// TIA Portal V17 export
// export: Created 2023-12-22T15:05:31.7217918Z, ExportSetting WithDefaults, DisplayName Totally Integrated Automation Portal, DisplayVersion V17, DisplayName TIA Portal Openness, DisplayVersion V17, DisplayName TIA Portal Version Control Interface, DisplayVersion V17, DisplayName STEP 7 Professional, DisplayVersion V17, DisplayName STEP 7 Safety, DisplayVersion V17, DisplayName WinCC Advanced, DisplayVersion V17
FUNCTION_BLOCK "FB_DRV_Start"   // FB100, LAD
{ S7_Optimized_Access := 'TRUE' }
VERSION : 0.1
// stored: AutoNumber false, IsIECCheckEnabled false, IsRetainMemResEnabled false, MemoryReserve 100, SetENOAutomatically false, UDAEnableTagReadback false
   VAR
      last_01s : Int;
      last_05s : Int;
      last_1s : Int;
      last_5s : Int;
      last_10s : Int;
      last_30s : Int;
      last_1m : Int;
      last_5m : Int;
      last_10m : Int;
      last_30m : Int;
      last_1h : Int;
      last_1_day : Int;
      last_1_week : Int;
      last_1_month : Int;
      last_s1 : Int;
      last_s2 : Int;
      "1h_minutes" { S7_SetPoint := 'True'} : Int;
      "1_day_hour" { S7_SetPoint := 'True'} : Int;
      "1_day_minutes" { S7_SetPoint := 'True'} : Int;
      "1_week_weekday" { S7_SetPoint := 'True'} : Int := 1;
      "1_week_hour" { S7_SetPoint := 'True'} : Int;
      "1_week_minutes" { S7_SetPoint := 'True'} : Int;
      "1_month_date" { S7_SetPoint := 'True'} : Int := 1;
      "1_month_hour" { S7_SetPoint := 'True'} : Int;
      "1_month_minutes" { S7_SetPoint := 'True'} : Int;
      s1_hour : Int := 8;
      s1_minutes : Int;
      s2_hour : Int := 20;
      s2_minutes : Int;
      pos : Array[0..15] of Bool;
      Error : Word;
      x { S7_SetPoint := 'True'} : "Protection";
   END_VAR
   VAR_TEMP
      cnt_01s : Int;
      cnt_5s : Int;
      cnt_10s : Int;
      cnt_30s : Int;
      cnt_5m : Int;
      cnt_10m : Int;
      cnt_30m : Int;
   END_VAR
   VAR_TEMP   // added for the SCL form of the ladder/FBD networks
      _w1 : Bool;
      _w2 : Bool;
   END_VAR
BEGIN

REGION Network 1: Обработчик системного времени
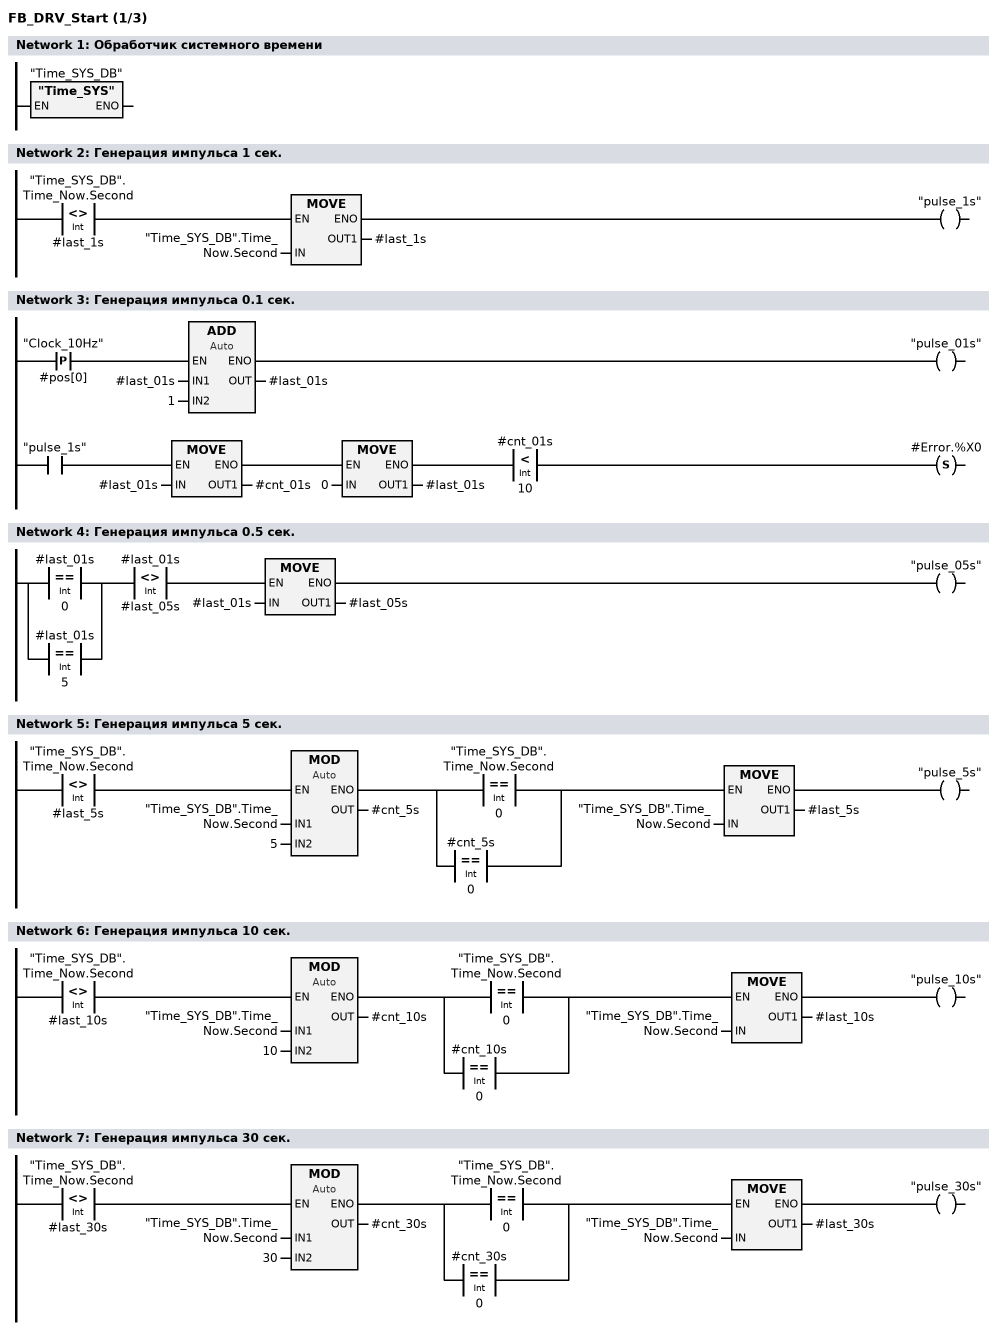
   RUNG wire#powerrail
      "Time_SYS_DB"()
   END_RUNG
   // the same network as SCL:
   "Time_SYS_DB"();   // "Time_SYS"
END_REGION

REGION Network 2: Генерация импульса 1 сек.
   RUNG wire#powerrail
      { S7_Templates := "SrcType := Int" } NE_Contact(in1 := "Time_SYS_DB".Time_Now.Second, in2 := #last_1s)
      Move(in := "Time_SYS_DB".Time_Now.Second, out1 => #last_1s)
      Coil( "pulse_1s" )
   END_RUNG
   // the same network as SCL:
   #_w1 := "Time_SYS_DB".Time_Now.Second <> #last_1s;
   IF #_w1 THEN #last_1s := "Time_SYS_DB".Time_Now.Second; END_IF;
   "pulse_1s" := #_w1;
END_REGION

REGION Network 3: Генерация импульса 0.1 сек.
   RUNG wire#powerrail
      P_Contact(operand := "Clock_10Hz", bit := #pos[0])
      Add(in1 := #last_01s, in2 := 1, out => #last_01s)
      Coil( "pulse_01s" )
   END_RUNG
   RUNG wire#powerrail
      Contact( "pulse_1s" )
      Move(in := #last_01s, out1 => #cnt_01s)
      Move(in := 0, out1 => #last_01s)
      { S7_Templates := "SrcType := Int" } LT_Contact(in1 := #cnt_01s, in2 := 10)
      S_Coil( #Error.%X0 )
   END_RUNG
   // the same network as SCL:
   #_w1 := "Clock_10Hz" AND NOT #pos[0];   // rising edge of "Clock_10Hz"
   #pos[0] := "Clock_10Hz";
   IF #_w1 THEN #last_01s := #last_01s + 1; END_IF;
   "pulse_01s" := #_w1;
   IF "pulse_1s" THEN
       #cnt_01s := #last_01s;
       #last_01s := 0;
   END_IF;
   IF "pulse_1s" AND (#cnt_01s < 10) THEN #Error.%X0 := TRUE; END_IF;
END_REGION

REGION Network 4: Генерация импульса 0.5 сек.
   RUNG wire#powerrail
      { S7_Templates := "SrcType := Int" } EQ_Contact(in1 := #last_01s, in2 := 0)
      wire#w1
      { S7_Templates := "SrcType := Int" } NE_Contact(in1 := #last_01s, in2 := #last_05s)
      Move(in := #last_01s, out1 => #last_05s)
      Coil( "pulse_05s" )
   END_RUNG
   RUNG wire#powerrail
      { S7_Templates := "SrcType := Int" } EQ_Contact(in1 := #last_01s, in2 := 5)
   END_RUNG wire#w1
   // the same network as SCL:
   #_w1 := ((#last_01s = 0) OR (#last_01s = 5)) AND (#last_01s <> #last_05s);
   IF #_w1 THEN #last_05s := #last_01s; END_IF;
   "pulse_05s" := #_w1;
END_REGION

REGION Network 5: Генерация импульса 5 сек.
   RUNG wire#powerrail
      { S7_Templates := "SrcType := Int" } NE_Contact(in1 := "Time_SYS_DB".Time_Now.Second, in2 := #last_5s)
      Mod(in1 := "Time_SYS_DB".Time_Now.Second, in2 := 5, out => #cnt_5s)
      wire#w1
      { S7_Templates := "SrcType := Int" } EQ_Contact(in1 := "Time_SYS_DB".Time_Now.Second, in2 := 0)
      wire#w2
      Move(in := "Time_SYS_DB".Time_Now.Second, out1 => #last_5s)
      Coil( "pulse_5s" )
   END_RUNG
   RUNG wire#w1
      { S7_Templates := "SrcType := Int" } EQ_Contact(in1 := #cnt_5s, in2 := 0)
   END_RUNG wire#w2
   // the same network as SCL:
   #_w1 := "Time_SYS_DB".Time_Now.Second <> #last_5s;
   IF #_w1 THEN #cnt_5s := "Time_SYS_DB".Time_Now.Second MOD 5; END_IF;
   #_w2 := #_w1 AND (("Time_SYS_DB".Time_Now.Second = 0) OR (#cnt_5s = 0));
   IF #_w2 THEN #last_5s := "Time_SYS_DB".Time_Now.Second; END_IF;
   "pulse_5s" := #_w2;
END_REGION

REGION Network 6: Генерация импульса 10 сек.
   RUNG wire#powerrail
      { S7_Templates := "SrcType := Int" } NE_Contact(in1 := "Time_SYS_DB".Time_Now.Second, in2 := #last_10s)
      Mod(in1 := "Time_SYS_DB".Time_Now.Second, in2 := 10, out => #cnt_10s)
      wire#w1
      { S7_Templates := "SrcType := Int" } EQ_Contact(in1 := "Time_SYS_DB".Time_Now.Second, in2 := 0)
      wire#w2
      Move(in := "Time_SYS_DB".Time_Now.Second, out1 => #last_10s)
      Coil( "pulse_10s" )
   END_RUNG
   RUNG wire#w1
      { S7_Templates := "SrcType := Int" } EQ_Contact(in1 := #cnt_10s, in2 := 0)
   END_RUNG wire#w2
   // the same network as SCL:
   #_w1 := "Time_SYS_DB".Time_Now.Second <> #last_10s;
   IF #_w1 THEN #cnt_10s := "Time_SYS_DB".Time_Now.Second MOD 10; END_IF;
   #_w2 := #_w1 AND (("Time_SYS_DB".Time_Now.Second = 0) OR (#cnt_10s = 0));
   IF #_w2 THEN #last_10s := "Time_SYS_DB".Time_Now.Second; END_IF;
   "pulse_10s" := #_w2;
END_REGION

REGION Network 7: Генерация импульса 30 сек.
   RUNG wire#powerrail
      { S7_Templates := "SrcType := Int" } NE_Contact(in1 := "Time_SYS_DB".Time_Now.Second, in2 := #last_30s)
      Mod(in1 := "Time_SYS_DB".Time_Now.Second, in2 := 30, out => #cnt_30s)
      wire#w1
      { S7_Templates := "SrcType := Int" } EQ_Contact(in1 := "Time_SYS_DB".Time_Now.Second, in2 := 0)
      wire#w2
      Move(in := "Time_SYS_DB".Time_Now.Second, out1 => #last_30s)
      Coil( "pulse_30s" )
   END_RUNG
   RUNG wire#w1
      { S7_Templates := "SrcType := Int" } EQ_Contact(in1 := #cnt_30s, in2 := 0)
   END_RUNG wire#w2
   // the same network as SCL:
   #_w1 := "Time_SYS_DB".Time_Now.Second <> #last_30s;
   IF #_w1 THEN #cnt_30s := "Time_SYS_DB".Time_Now.Second MOD 30; END_IF;
   #_w2 := #_w1 AND (("Time_SYS_DB".Time_Now.Second = 0) OR (#cnt_30s = 0));
   IF #_w2 THEN #last_30s := "Time_SYS_DB".Time_Now.Second; END_IF;
   "pulse_30s" := #_w2;
END_REGION

REGION Network 8: Генерация импульса 1 мин.
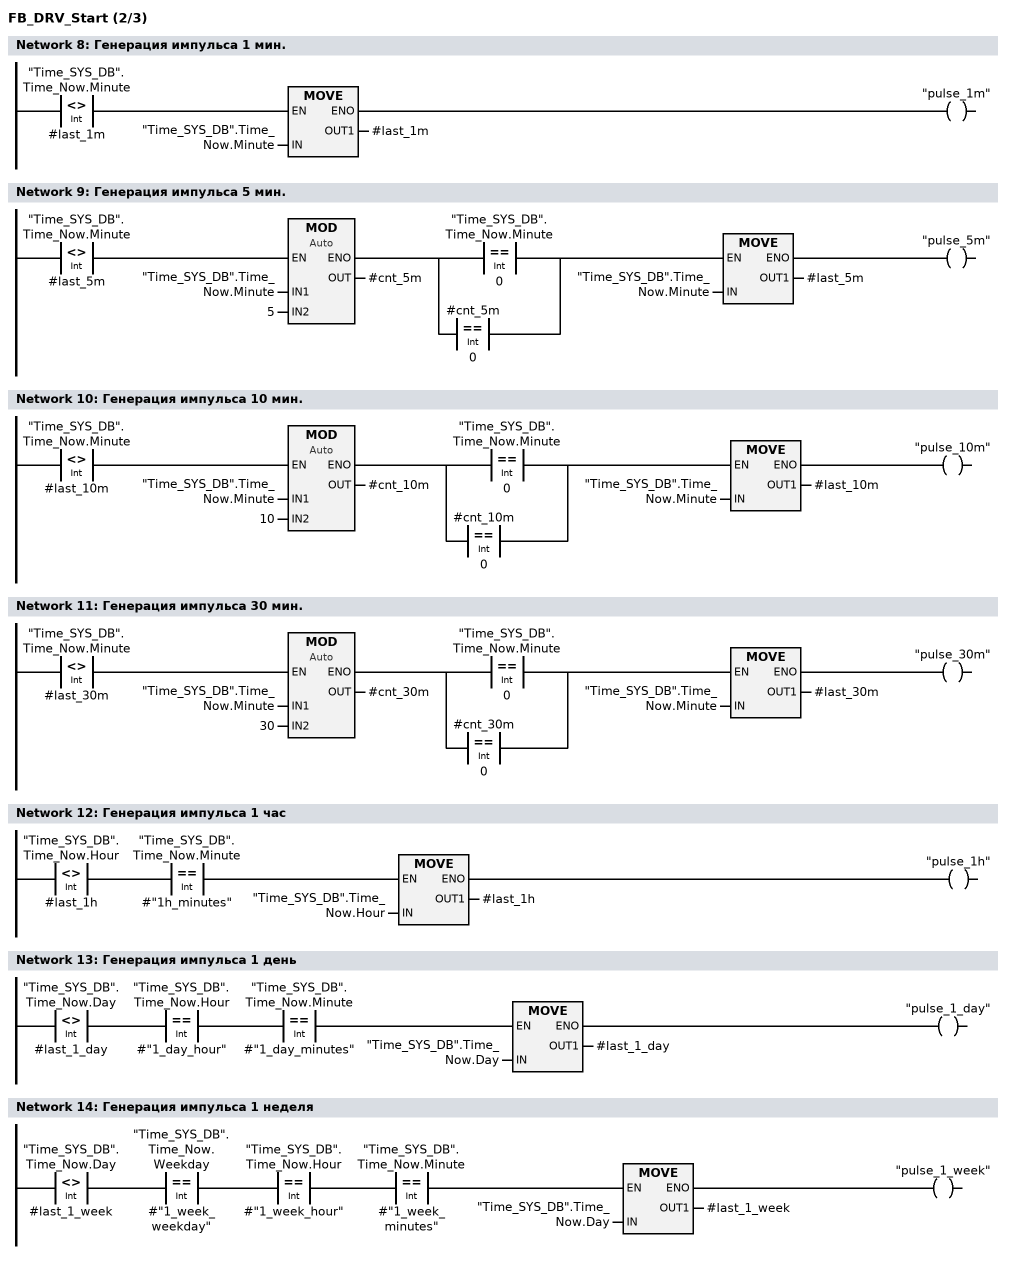
   RUNG wire#powerrail
      { S7_Templates := "SrcType := Int" } NE_Contact(in1 := "Time_SYS_DB".Time_Now.Minute, in2 := #last_1m)
      Move(in := "Time_SYS_DB".Time_Now.Minute, out1 => #last_1m)
      Coil( "pulse_1m" )
   END_RUNG
   // the same network as SCL:
   #_w1 := "Time_SYS_DB".Time_Now.Minute <> #last_1m;
   IF #_w1 THEN #last_1m := "Time_SYS_DB".Time_Now.Minute; END_IF;
   "pulse_1m" := #_w1;
END_REGION

REGION Network 9: Генерация импульса 5 мин.
   RUNG wire#powerrail
      { S7_Templates := "SrcType := Int" } NE_Contact(in1 := "Time_SYS_DB".Time_Now.Minute, in2 := #last_5m)
      Mod(in1 := "Time_SYS_DB".Time_Now.Minute, in2 := 5, out => #cnt_5m)
      wire#w1
      { S7_Templates := "SrcType := Int" } EQ_Contact(in1 := "Time_SYS_DB".Time_Now.Minute, in2 := 0)
      wire#w2
      Move(in := "Time_SYS_DB".Time_Now.Minute, out1 => #last_5m)
      Coil( "pulse_5m" )
   END_RUNG
   RUNG wire#w1
      { S7_Templates := "SrcType := Int" } EQ_Contact(in1 := #cnt_5m, in2 := 0)
   END_RUNG wire#w2
   // the same network as SCL:
   #_w1 := "Time_SYS_DB".Time_Now.Minute <> #last_5m;
   IF #_w1 THEN #cnt_5m := "Time_SYS_DB".Time_Now.Minute MOD 5; END_IF;
   #_w2 := #_w1 AND (("Time_SYS_DB".Time_Now.Minute = 0) OR (#cnt_5m = 0));
   IF #_w2 THEN #last_5m := "Time_SYS_DB".Time_Now.Minute; END_IF;
   "pulse_5m" := #_w2;
END_REGION

REGION Network 10: Генерация импульса 10 мин.
   RUNG wire#powerrail
      { S7_Templates := "SrcType := Int" } NE_Contact(in1 := "Time_SYS_DB".Time_Now.Minute, in2 := #last_10m)
      Mod(in1 := "Time_SYS_DB".Time_Now.Minute, in2 := 10, out => #cnt_10m)
      wire#w1
      { S7_Templates := "SrcType := Int" } EQ_Contact(in1 := "Time_SYS_DB".Time_Now.Minute, in2 := 0)
      wire#w2
      Move(in := "Time_SYS_DB".Time_Now.Minute, out1 => #last_10m)
      Coil( "pulse_10m" )
   END_RUNG
   RUNG wire#w1
      { S7_Templates := "SrcType := Int" } EQ_Contact(in1 := #cnt_10m, in2 := 0)
   END_RUNG wire#w2
   // the same network as SCL:
   #_w1 := "Time_SYS_DB".Time_Now.Minute <> #last_10m;
   IF #_w1 THEN #cnt_10m := "Time_SYS_DB".Time_Now.Minute MOD 10; END_IF;
   #_w2 := #_w1 AND (("Time_SYS_DB".Time_Now.Minute = 0) OR (#cnt_10m = 0));
   IF #_w2 THEN #last_10m := "Time_SYS_DB".Time_Now.Minute; END_IF;
   "pulse_10m" := #_w2;
END_REGION

REGION Network 11: Генерация импульса 30 мин.
   RUNG wire#powerrail
      { S7_Templates := "SrcType := Int" } NE_Contact(in1 := "Time_SYS_DB".Time_Now.Minute, in2 := #last_30m)
      Mod(in1 := "Time_SYS_DB".Time_Now.Minute, in2 := 30, out => #cnt_30m)
      wire#w1
      { S7_Templates := "SrcType := Int" } EQ_Contact(in1 := "Time_SYS_DB".Time_Now.Minute, in2 := 0)
      wire#w2
      Move(in := "Time_SYS_DB".Time_Now.Minute, out1 => #last_30m)
      Coil( "pulse_30m" )
   END_RUNG
   RUNG wire#w1
      { S7_Templates := "SrcType := Int" } EQ_Contact(in1 := #cnt_30m, in2 := 0)
   END_RUNG wire#w2
   // the same network as SCL:
   #_w1 := "Time_SYS_DB".Time_Now.Minute <> #last_30m;
   IF #_w1 THEN #cnt_30m := "Time_SYS_DB".Time_Now.Minute MOD 30; END_IF;
   #_w2 := #_w1 AND (("Time_SYS_DB".Time_Now.Minute = 0) OR (#cnt_30m = 0));
   IF #_w2 THEN #last_30m := "Time_SYS_DB".Time_Now.Minute; END_IF;
   "pulse_30m" := #_w2;
END_REGION

REGION Network 12: Генерация импульса 1 час
   RUNG wire#powerrail
      { S7_Templates := "SrcType := Int" } NE_Contact(in1 := "Time_SYS_DB".Time_Now.Hour, in2 := #last_1h)
      { S7_Templates := "SrcType := Int" } EQ_Contact(in1 := "Time_SYS_DB".Time_Now.Minute, in2 := #"1h_minutes")
      Move(in := "Time_SYS_DB".Time_Now.Hour, out1 => #last_1h)
      Coil( "pulse_1h" )
   END_RUNG
   // the same network as SCL:
   #_w1 := ("Time_SYS_DB".Time_Now.Hour <> #last_1h) AND ("Time_SYS_DB".Time_Now.Minute = #"1h_minutes");
   IF #_w1 THEN #last_1h := "Time_SYS_DB".Time_Now.Hour; END_IF;
   "pulse_1h" := #_w1;
END_REGION

REGION Network 13: Генерация импульса 1 день
   RUNG wire#powerrail
      { S7_Templates := "SrcType := Int" } NE_Contact(in1 := "Time_SYS_DB".Time_Now.Day, in2 := #last_1_day)
      { S7_Templates := "SrcType := Int" } EQ_Contact(in1 := "Time_SYS_DB".Time_Now.Hour, in2 := #"1_day_hour")
      { S7_Templates := "SrcType := Int" } EQ_Contact(in1 := "Time_SYS_DB".Time_Now.Minute, in2 := #"1_day_minutes")
      Move(in := "Time_SYS_DB".Time_Now.Day, out1 => #last_1_day)
      Coil( "pulse_1_day" )
   END_RUNG
   // the same network as SCL:
   #_w1 := ("Time_SYS_DB".Time_Now.Day <> #last_1_day) AND ("Time_SYS_DB".Time_Now.Hour = #"1_day_hour") AND ("Time_SYS_DB".Time_Now.Minute = #"1_day_minutes");
   IF #_w1 THEN #last_1_day := "Time_SYS_DB".Time_Now.Day; END_IF;
   "pulse_1_day" := #_w1;
END_REGION

REGION Network 14: Генерация импульса 1 неделя
   RUNG wire#powerrail
      { S7_Templates := "SrcType := Int" } NE_Contact(in1 := "Time_SYS_DB".Time_Now.Day, in2 := #last_1_week)
      { S7_Templates := "SrcType := Int" } EQ_Contact(in1 := "Time_SYS_DB".Time_Now.Weekday, in2 := #"1_week_weekday")
      { S7_Templates := "SrcType := Int" } EQ_Contact(in1 := "Time_SYS_DB".Time_Now.Hour, in2 := #"1_week_hour")
      { S7_Templates := "SrcType := Int" } EQ_Contact(in1 := "Time_SYS_DB".Time_Now.Minute, in2 := #"1_week_minutes")
      Move(in := "Time_SYS_DB".Time_Now.Day, out1 => #last_1_week)
      Coil( "pulse_1_week" )
   END_RUNG
   // the same network as SCL:
   #_w1 := ("Time_SYS_DB".Time_Now.Day <> #last_1_week) AND ("Time_SYS_DB".Time_Now.Weekday = #"1_week_weekday") AND ("Time_SYS_DB".Time_Now.Hour = #"1_week_hour") AND ("Time_SYS_DB".Time_Now.Minute = #"1_week_minutes");
   IF #_w1 THEN #last_1_week := "Time_SYS_DB".Time_Now.Day; END_IF;
   "pulse_1_week" := #_w1;
END_REGION

REGION Network 15: Генерация импульса 1 месяц
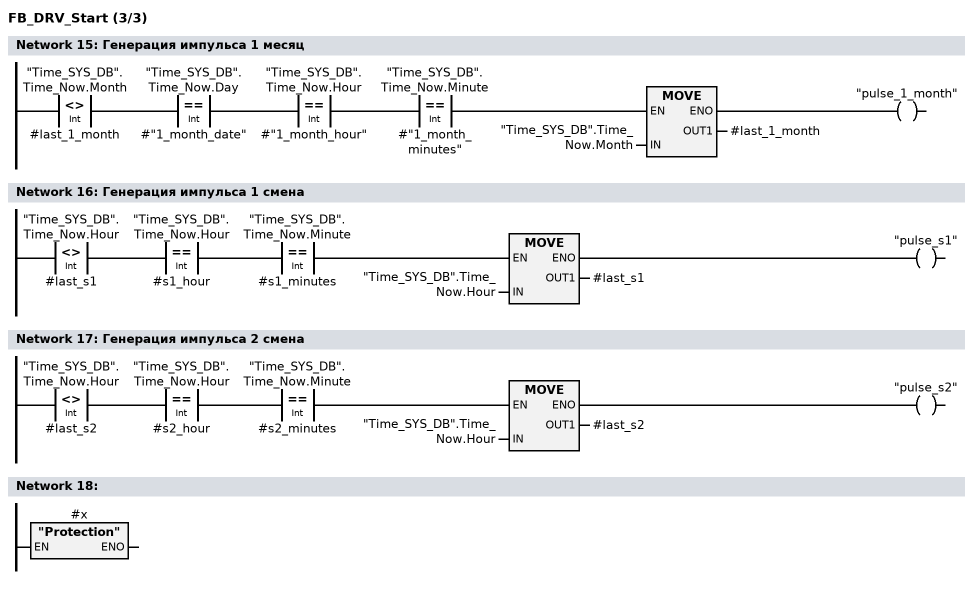
   RUNG wire#powerrail
      { S7_Templates := "SrcType := Int" } NE_Contact(in1 := "Time_SYS_DB".Time_Now.Month, in2 := #last_1_month)
      { S7_Templates := "SrcType := Int" } EQ_Contact(in1 := "Time_SYS_DB".Time_Now.Day, in2 := #"1_month_date")
      { S7_Templates := "SrcType := Int" } EQ_Contact(in1 := "Time_SYS_DB".Time_Now.Hour, in2 := #"1_month_hour")
      { S7_Templates := "SrcType := Int" } EQ_Contact(in1 := "Time_SYS_DB".Time_Now.Minute, in2 := #"1_month_minutes")
      Move(in := "Time_SYS_DB".Time_Now.Month, out1 => #last_1_month)
      Coil( "pulse_1_month" )
   END_RUNG
   // the same network as SCL:
   #_w1 := ("Time_SYS_DB".Time_Now.Month <> #last_1_month) AND ("Time_SYS_DB".Time_Now.Day = #"1_month_date") AND ("Time_SYS_DB".Time_Now.Hour = #"1_month_hour") AND ("Time_SYS_DB".Time_Now.Minute = #"1_month_minutes");
   IF #_w1 THEN #last_1_month := "Time_SYS_DB".Time_Now.Month; END_IF;
   "pulse_1_month" := #_w1;
END_REGION

REGION Network 16: Генерация импульса 1 смена
   RUNG wire#powerrail
      { S7_Templates := "SrcType := Int" } NE_Contact(in1 := "Time_SYS_DB".Time_Now.Hour, in2 := #last_s1)
      { S7_Templates := "SrcType := Int" } EQ_Contact(in1 := "Time_SYS_DB".Time_Now.Hour, in2 := #s1_hour)
      { S7_Templates := "SrcType := Int" } EQ_Contact(in1 := "Time_SYS_DB".Time_Now.Minute, in2 := #s1_minutes)
      Move(in := "Time_SYS_DB".Time_Now.Hour, out1 => #last_s1)
      Coil( "pulse_s1" )
   END_RUNG
   // the same network as SCL:
   #_w1 := ("Time_SYS_DB".Time_Now.Hour <> #last_s1) AND ("Time_SYS_DB".Time_Now.Hour = #s1_hour) AND ("Time_SYS_DB".Time_Now.Minute = #s1_minutes);
   IF #_w1 THEN #last_s1 := "Time_SYS_DB".Time_Now.Hour; END_IF;
   "pulse_s1" := #_w1;
END_REGION

REGION Network 17: Генерация импульса 2 смена
   RUNG wire#powerrail
      { S7_Templates := "SrcType := Int" } NE_Contact(in1 := "Time_SYS_DB".Time_Now.Hour, in2 := #last_s2)
      { S7_Templates := "SrcType := Int" } EQ_Contact(in1 := "Time_SYS_DB".Time_Now.Hour, in2 := #s2_hour)
      { S7_Templates := "SrcType := Int" } EQ_Contact(in1 := "Time_SYS_DB".Time_Now.Minute, in2 := #s2_minutes)
      Move(in := "Time_SYS_DB".Time_Now.Hour, out1 => #last_s2)
      Coil( "pulse_s2" )
   END_RUNG
   // the same network as SCL:
   #_w1 := ("Time_SYS_DB".Time_Now.Hour <> #last_s2) AND ("Time_SYS_DB".Time_Now.Hour = #s2_hour) AND ("Time_SYS_DB".Time_Now.Minute = #s2_minutes);
   IF #_w1 THEN #last_s2 := "Time_SYS_DB".Time_Now.Hour; END_IF;
   "pulse_s2" := #_w1;
END_REGION

REGION Network 18
   RUNG wire#powerrail
      #x()
   END_RUNG
   // the same network as SCL:
   #x();   // "Protection"
END_REGION
END_FUNCTION_BLOCK
